FUNCTION_BLOCK SHAFT_MDL (* Model for a Rotating Shaft *)
  (* Standard: 61499-1 *)
  (* Version 0.3, 2004-09-04, JHC, Rockwell Automation, Subclassed from E_CYCLE. *)
  (* Version 0.2, 2001-04-24, JHC, Rockwell Automation, Moved to fb.rt.process. *)
  (* Version 0.1, 2000-06-21, JHC, Rockwell Automation, Uses LibraryElement.dtd *)
  (* Version 0.0, 2000-05-01, JHC, Rockwell Automation *)
  (* Compiler header: package fb.rt.process; *)
  (* Compiler classdef: public class SHAFT_MDL extends E_CYCLE *)
  (* Compiler Java Sun JDK 1.4.2 *)
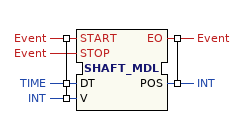
  EVENT_INPUT
    START WITH DT, V; (* Start Model *)
    STOP; (* Stop Model *)
  END_EVENT
  EVENT_OUTPUT
    EO WITH POS; (* Update POS *)
  END_EVENT
  VAR_INPUT
    DT : TIME; (* Simulation Time Increment *)
    V : INT; (* Angular velocity, degrees per second *)
  END_VAR
  VAR_OUTPUT
    POS : INT; (* Pump Shaft Position {-359 to +359 degrees} *)
  END_VAR
END_FUNCTION_BLOCK
